FUNCTION_BLOCK E_TRAIN (* Generate of a finite train of events seperated by the time DT *)
  (* Standard: 61499-1 Annex A; Description: Copyright (c) 2017 fortiss GmbH This program and the accompanying materials are made available under the terms of the Eclipse Public License 2.0 which is available at https://www.eclipse.org/legal/epl-2.0/ SPDX-License-Identifier: EPL-2.0 *)
  (* Version 1.0, 2017-09-22, Alois Zoitl, fortiss GmbH, initial API and implementation and/or initial documentation *)
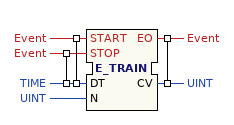
  EVENT_INPUT
    START WITH DT; (* Start event generation *)
    STOP WITH DT; (* Stop event generation *)
  END_EVENT
  EVENT_OUTPUT
    EO WITH CV; (* Generated events *)
  END_EVENT
  VAR_INPUT
    DT : TIME; (* Time by which the events should be seperated *)
    N : UINT; (* Number of events to generate *)
  END_VAR
  VAR_OUTPUT
    CV : UINT; (* count of the current event: EO index (0..N-1) *)
  END_VAR
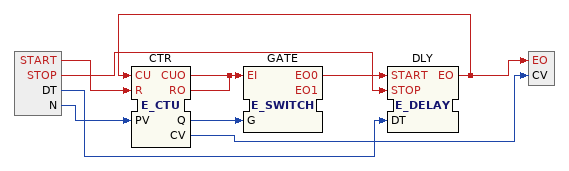
  FBS
    CTR : E_CTU;
    GATE : E_SWITCH;
    DLY : E_DELAY;
  END_FBS
  EVENT_CONNECTIONS
    CTR.CUO TO GATE.EI;
    CTR.RO TO GATE.EI;
    START TO CTR.R;
    GATE.EO0 TO DLY.START;
    STOP TO DLY.STOP;
    DLY.EO TO EO;
    DLY.EO TO CTR.CU;
  END_CONNECTIONS
  DATA_CONNECTIONS
    N TO CTR.PV;
    CTR.CV TO CV;
    DT TO DLY.DT;
    CTR.Q TO GATE.G;
  END_CONNECTIONS
END_FUNCTION_BLOCK
